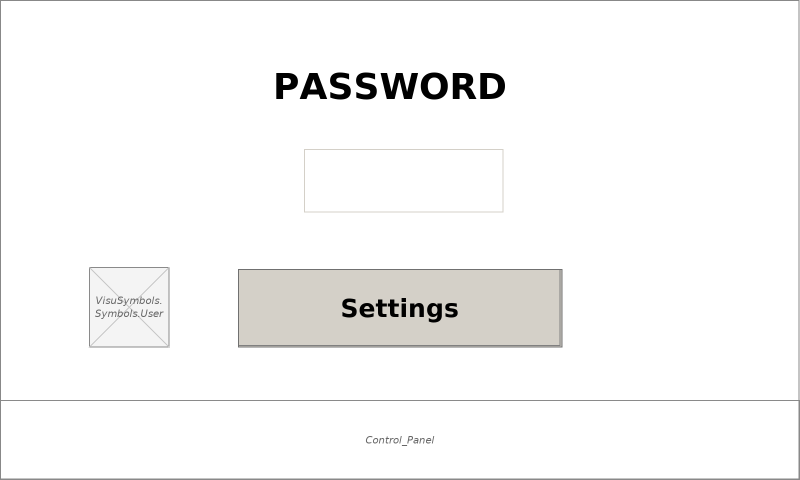
VISUALIZATION Password  // 800x480
    Frame (0,400 800x80)
        shows Control_Panel()
    Label (233,35 289x103), "PASSWORD"
    Textfield (304,149 199x63), text variable: GVL_IO.Password_IN
        OnMouseClick: write the text variable via Default, password
    Button (238,269 324x78), "Settings", invisible if: GVL_IO.Password_IN <> 9118
        OnMouseClick: change screen: Settings
    Image (89,267 80x80), invisible if: GVL_IO.Password_IN <> 9118, image: VisuSymbols.Symbols.User
        OnMouseClick: change screen: Overview
END_VISUALIZATION

(* stored: Version 1.1.0.1, ProductVersion 3.1.4024.13
   Visu Password: Id {e3b4d4f7-6319-4b57-a0a5-dbb82a51d9d2} *)
